FUNCTION_BLOCK FB_LinearActuator
VAR
    bEnable          : BOOL;         
END_VAR

VAR_INPUT
	bRelayForward    : POINTER TO BOOL; 
    bRelayReverse    : POINTER TO BOOL; 
END_VAR

METHOD Enable : BOOL
VAR_INPUT
    bEnableCmd : BOOL;
END_VAR
bEnable := bEnableCmd;
IF NOT bEnable THEN

	bRelayForward^ := FALSE;
	bRelayReverse^ := FALSE;
END_IF;
Enable := bEnable;
END_METHOD

METHOD FB_init : BOOL
VAR_INPUT
  bInitRetains : BOOL;
  bInCopyCode  : BOOL;
END_VAR

FB_init := TRUE;
END_METHOD

METHOD MoveForward : BOOL
VAR_INPUT
    bStart : BOOL;
END_VAR
IF bEnable THEN
	bRelayForward^ := bStart;  
	bRelayReverse^ := FALSE;   
	MoveForward := bStart;
ELSE
	MoveForward := FALSE;
END_IF;
END_METHOD

METHOD MoveReverse : BOOL
VAR_INPUT
    bStart : BOOL;
END_VAR
IF bEnable THEN
	bRelayReverse^ := bStart;  
	bRelayForward^ := FALSE;   
	MoveReverse := bStart;
ELSE
	MoveReverse := FALSE;
END_IF;
END_METHOD

METHOD Stop : BOOL
VAR_INPUT
END_VAR

bRelayForward^ := FALSE;
bRelayReverse^ := FALSE;
Stop := TRUE;
END_METHOD

END_FUNCTION_BLOCK

(* stored: Version 1.1.0.1, ProductVersion 3.1.4024.14
   POU FB_LinearActuator: Id {ea18bd47-f142-4882-be0a-b1771c69605b}, SpecialFunc None
   Method Enable: Id {5781204b-ff90-43fa-8680-a505886ae8fc}
   Method FB_init: Id {97589f9e-12e3-42ec-a9fa-23e9e6bb3543}
   Method MoveForward: Id {05889208-3945-4579-8e80-ba06223a15bb}
   Method MoveReverse: Id {fc96ee79-2f9e-44d9-b4a7-e028c83a156a}
   Method Stop: Id {ed4bc20c-08fd-49e2-8da7-e700d0af9ca8} *)
